Omron CX-Programmer project NewProject (CX-Programmer 9.54)

# PLC Automation_project_station4: CJ1M CPU11

## Global symbols (name address type ; comment)
0.00 BOOL  ; Start_PB
0.01 BOOL  ; Stop_PB
0.02 BOOL  ; Reset_PB
0.03 BOOL  ; Emergency_PB
0.04 BOOL  ; Palletizer  Pusher Limit
0.05 BOOL  ; Box Conveyor
0.06 BOOL  ; Box Conveyor Incline
0.07 BOOL  ; Diff_Sensor1
0.08 BOOL  ; Diff_Sensor 2
0.13 BOOL  ; Diff_Sensor 1
0.14 BOOL  ; Diff_Sensor
1.00 BOOL  ; Status
1.01 BOOL  ; Start_Light
1.02 BOOL  ; Start Light
1.03 BOOL  ; Stop_Light
1.04 BOOL  ; Reset Light
1.05 BOOL  ; Box Conveyor
1.06 BOOL  ; Box Conveyor Incline
1.07 BOOL  ; Roller Stop In
1.08 BOOL  ; Patellizer Pusher
1.09 BOOL  ; Palletizer Plate Open
1.10 BOOL  ; Roller Stop Out
1.11 BOOL  ; Receiver Box Conveyor in
1.12 BOOL  ; Receiver Box Conveyor Inclined Out
1.13 BOOL  ; Palletizing Box Emitter
1.14 BOOL  ; Palletizer Conveyor
1.15 BOOL  ; Stackable_Box_Emitter
D10 CHANNEL  ; Palletizing Box Counting
D11 CHANNEL  ; Stackable Box Counting
T0002 BOOL  ; 4
T0004 BOOL  ; #20
W10.00 BOOL  ; Roller_Stopper_In_Control
W10.01 BOOL  ; Roller_Stopper_Out_Control
W10.02 BOOL  ; Reset Counting
W1.00 BOOL  ; Status
W1.01 BOOL  ; Emergency_Status
W20.00 BOOL  ; Pusher_Control

## Program NewProgram1 (cyclic task 0)

### Section Section1

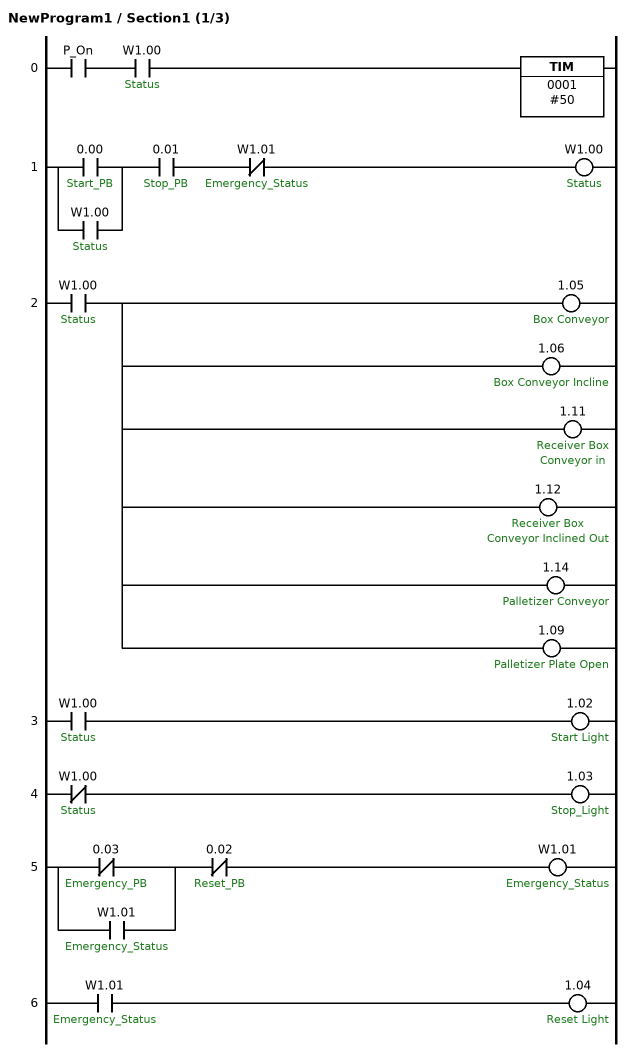
; rung 0
LD P_On
AND W1.00  ; Status
TIM 0001 #50
; rung 1
LD 0.00  ; Start_PB
OR W1.00  ; Status
AND 0.01  ; Stop_PB
ANDNOT W1.01  ; Emergency_Status
OUT W1.00  ; Status
; rung 2
LD W1.00  ; Status
OUT 1.05  ; Box Conveyor
OUT 1.06  ; Box Conveyor Incline
OUT 1.11  ; Receiver Box Conveyor in
OUT 1.12  ; Receiver Box Conveyor Inclined Out
OUT 1.14  ; Palletizer Conveyor
OUT 1.09  ; Palletizer Plate Open
; rung 3
LD W1.00  ; Status
OUT 1.02  ; Start Light
; rung 4
LDNOT W1.00  ; Status
OUT 1.03  ; Stop_Light
; rung 5
LDNOT 0.03  ; Emergency_PB
OR W1.01  ; Emergency_Status
ANDNOT 0.02  ; Reset_PB
OUT W1.01  ; Emergency_Status
; rung 6
LD W1.01  ; Emergency_Status
OUT 1.04  ; Reset Light

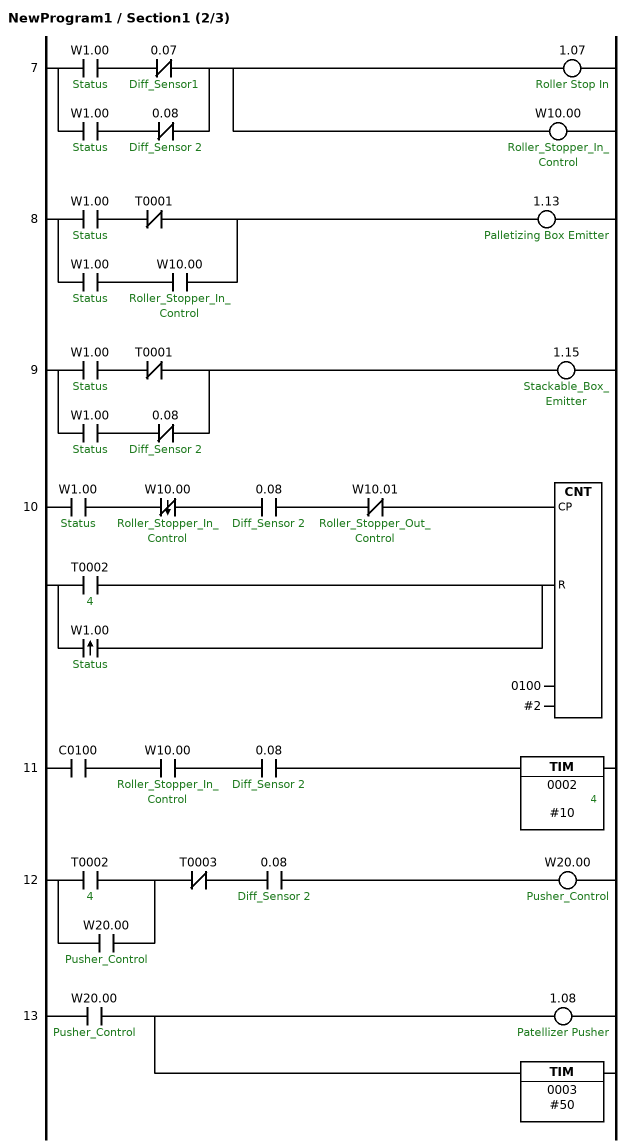
; rung 7
LD W1.00  ; Status
ANDNOT 0.07  ; Diff_Sensor1
LD W1.00  ; Status
ANDNOT 0.08  ; Diff_Sensor 2
ORLD
OUT 1.07  ; Roller Stop In
OUT W10.00  ; Roller_Stopper_In_Control
; rung 8
LD W1.00  ; Status
ANDNOT T0001
LD W1.00  ; Status
AND W10.00  ; Roller_Stopper_In_Control
ORLD
OUT 1.13  ; Palletizing Box Emitter
; rung 9
LD W1.00  ; Status
ANDNOT T0001
LD W1.00  ; Status
ANDNOT 0.08  ; Diff_Sensor 2
ORLD
OUT 1.15  ; Stackable_Box_Emitter
; rung 10
LD W1.00  ; Status
%ANDNOT W10.00  ; Roller_Stopper_In_Control
AND 0.08  ; Diff_Sensor 2
ANDNOT W10.01  ; Roller_Stopper_Out_Control
LD T0002  ; 4
@OR W1.00  ; Status
CNT 0100 #2
; rung 11
LD C0100
AND W10.00  ; Roller_Stopper_In_Control
AND 0.08  ; Diff_Sensor 2
TIM 0002 #10  ; 4
; rung 12
LD T0002  ; 4
OR W20.00  ; Pusher_Control
ANDNOT T0003
AND 0.08  ; Diff_Sensor 2
OUT W20.00  ; Pusher_Control
; rung 13
LD W20.00  ; Pusher_Control
OUT 1.08  ; Patellizer Pusher
TIM 0003 #50

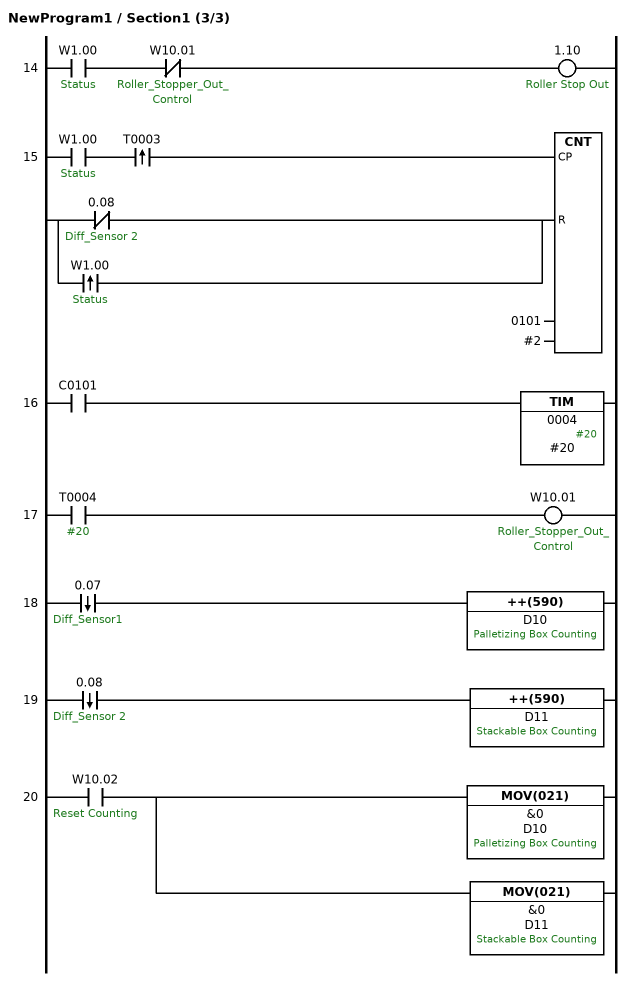
; rung 14
LD W1.00  ; Status
ANDNOT W10.01  ; Roller_Stopper_Out_Control
OUT 1.10  ; Roller Stop Out
; rung 15
LD W1.00  ; Status
@AND T0003
LDNOT 0.08  ; Diff_Sensor 2
@OR W1.00  ; Status
CNT 0101 #2
; rung 16
LD C0101
TIM 0004 #20  ; #20
; rung 17
LD T0004  ; #20
OUT W10.01  ; Roller_Stopper_Out_Control
; rung 18
%LD 0.07  ; Diff_Sensor1
++(590) D10  ; Palletizing Box Counting
; rung 19
%LD 0.08  ; Diff_Sensor 2
++(590) D11  ; Stackable Box Counting
; rung 20
LD W10.02  ; Reset Counting
MOV(021) &0 D10  ; Palletizing Box Counting
MOV(021) &0 D11  ; Stackable Box Counting

### Section END
; rung 0
END(001)